RoboDK station: Coursework_2.rdk

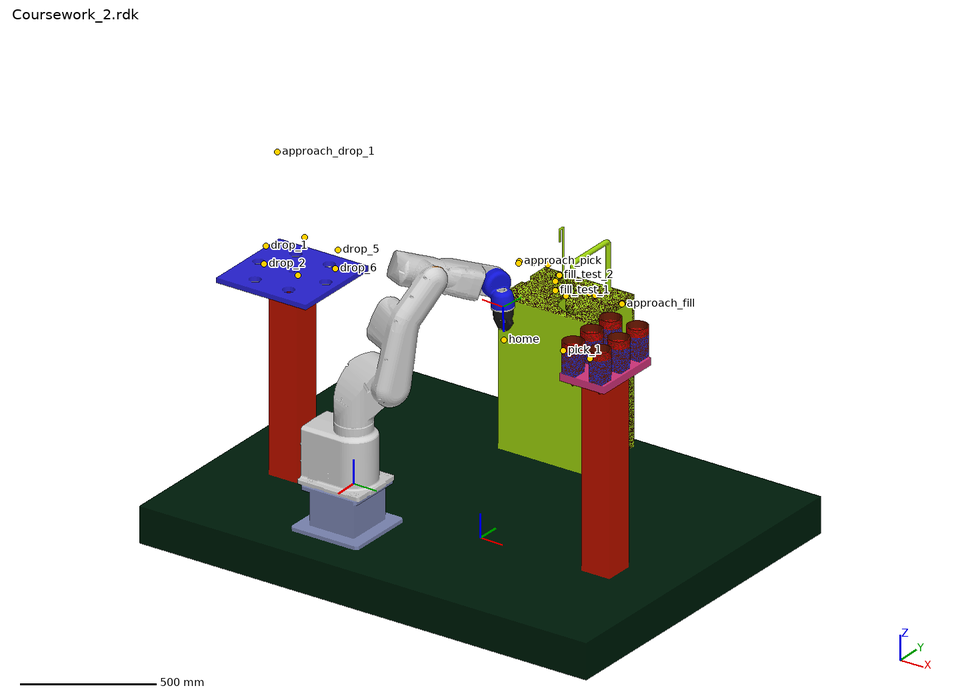
[picture v0: the station drawn from its stored meshes, robots at their saved joint values, targets as dots, program paths as lines]
Station Coursework_2 (saved by RoboDK 5.8.0). Poses are relative to the parent item; angles as X-Y-Z fixed-axis rotations.
Station parameters (name, value as stored): 153.91
  - frame Base_cell_frame at (0, 0, 0) mm
    - object PDE4431_CW2_2024 at (0, 0, 0) mm, rotated rx 90 ry 0 rz 0 deg, size 2000 x 980 x 1500 mm, geometry from PDE4431_CW2_2024.STEP
    - frame Epson VT6 Base at (-250, -450, 330) mm, rotated rx 0 ry 0 rz -90 deg
      - robot Epson VT6: 6 axes, payload 6 kg, reach 920 mm, repeatability 0.1 mm, weight 40 kg
          modified DH rows (alpha deg, a mm, theta deg, d mm): 0, 0, 0, 412; -90, 100, -90, 0; 0, 420, 0, 0; -90, 0, 0, 400; 90, 0, 0, 0; -90, 0, 0, 80
          base shift (0, 0, 0) mm, rotated rx 0 ry 0 rz 90 deg
          joint limits [-170, -160, -51, -200, -125, -360] to [170, 65, 190, 200, 125, 360]; home [0, 0, 0, 0, 0, 0]; saved at [66.458, -23.674, 0.501, 181.108, 64.729, -73.3]
        - frame RobotiQ 2F-140 Gripper (Mechanism) Base at (0, 0, 0) mm
          - robot RobotiQ 2F-140 Gripper (Mechanism) (model RobotiQ 2F140): 1 axes, payload 5 kg
              joint limits [0] to [140]; home [140]; saved at [99.47]
          - target open_gripper (Cartesian target) at (0, 0, 135) mm, rotated rx -90 ry 0 rz 90 deg; joints [99.47, 14.65, 163.72, -0.95, 89.45, -5.12] of RobotiQ 2F-140 Gripper (Mechanism)
          - target close_gripper (Cartesian target) at (0, 0, 135) mm, rotated rx -90 ry 0 rz 90 deg; joints [60, 27.47, -32.86, -122.29, -24.8, -148.93] of RobotiQ 2F-140 Gripper (Mechanism)
        - tool Tool 1, TCP at (0, 0, 135) mm, rotated rx -90 ry 0 rz 90 deg
      - object Pedestal_1 at (0, -30, -180) mm, rotated rx 90 ry 0 rz 0 deg, size 300 x 180 x 300 mm, geometry from Pedestal_1.STEP
    - frame input_table_frame at (0, 0, 0) mm
      - target home (Cartesian target) at (10.77, 139.13, 754.42) mm, rotated rx 88.42 ry -1.71 rz 83.64 deg; joints [-2.51, 19.29, -44.31, 1.89, -63.39, 85.3] of Epson VT6
      - target approach_pick (Cartesian target) at (397.26, -315.09, 1365.72) mm, rotated rx -100.11 ry -87.63 rz -171.58 deg; joints [18.089, -0.789, 29.967, 38.658, -32.785, 56.501] of Epson VT6
      - target pick_1 (Cartesian target) at (594.91, -318.66, 1058.51) mm, rotated rx -100.11 ry -87.63 rz -171.58 deg; joints [7.923, -20.29, 7.849, 146.461, -17.595, -57.734] of Epson VT6
      - target pick_2 (Cartesian target) at (715.78, -319.07, 1058.49) mm, rotated rx -126.16 ry -87.1 rz -145.13 deg; joints [6.525, -37.672, 34.127, 126.782, -9.811, -38.578] of Epson VT6
      - target approach_fill (Cartesian target) at (301.22, 477.28, 847.78) mm, rotated rx -50.46 ry -87.49 rz -131.29 deg; joints [-33.96, -23.408, -22.424, 40.243, 55.613, 64.831] of Epson VT6
      - target enter_fill (Cartesian target) at (181.46, 475.85, 849.63) mm, rotated rx -100.83 ry -88.03 rz -80.88 deg; joints [59.132, -56.563, 37.437, 56.856, 35.551, 37.301] of Epson VT6
      - target fill_1_go_down (Cartesian target) at (99.43, 408.13, 852.78) mm, rotated rx -100.83 ry -88.03 rz -80.88 deg; joints [61.936, -42.802, 12.032, 42.314, 41.214, 54.267] of Epson VT6
      - target fill_test_1 (Cartesian target) at (39.88, 425.07, 848.67) mm, rotated rx -100.83 ry -88.03 rz -80.88 deg; joints [66.768, -41.855, 9.609, 34.939, 39.793, 60.64] of Epson VT6
      - target approach_fill_2 (Cartesian target) at (-3.3, 486.34, 850.99) mm, rotated rx -100.83 ry -88.03 rz -80.88 deg; joints [71.584, -46.813, 19.15, 31.191, 33.677, 62.31] of Epson VT6
      - target fill_2_go_down (Cartesian target) at (-100.56, 579.23, 854.68) mm, rotated rx -100.83 ry -88.03 rz -80.88 deg; joints [79.404, -48.826, 23.503, 18.809, 28.583, 72.676] of Epson VT6
      - target fill_test (Cartesian target) at (-140.12, 595.57, 850.44) mm, rotated rx -100.83 ry -88.03 rz -80.88 deg; joints [82.903, -57.981, 40.297, 15.654, 20.323, 74.725] of Epson VT6
      - target fill_test_3 (Cartesian target) at (-161.01, 566.2, 849.56) mm, rotated rx -100.83 ry -88.03 rz -80.88 deg; joints [84.119, -53.062, 30.713, 10.031, 24.622, 80.354] of Epson VT6
      - target exit_fill (Cartesian target) at (-201.89, 537.42, 848.81) mm, rotated rx -100.83 ry -88.03 rz -80.88 deg; joints [86.913, -48.679, 22.293, 2.884, 28.353, 87.045] of Epson VT6
      - target approach_drop_1 (Cartesian target) at (-801.01, -152.39, 1410.63) mm, rotated rx -121.97 ry -88.27 rz 29.1 deg; joints [139.545, -3.407, 40.97, 127.197, 49.933, -51.748] of Epson VT6
      - target drop_1 (Cartesian target) at (-813.15, -207.69, 1046.6) mm, rotated rx -121.97 ry -88.27 rz 29.1 deg; joints [152.488, 12.57, -28.659, 56.431, 30.004, 35.87] of Epson VT6
      - target drop_2 (Cartesian target) at (-731.62, -336.84, 1047.6) mm, rotated rx -102.73 ry -87.66 rz 14.29 deg; joints [155.972, 28.648, -38.95, 65.094, 28.402, 26.221] of Epson VT6
      - target drop_3 (Cartesian target) at (-739.03, -66.95, 1045.18) mm, rotated rx -102.73 ry -87.66 rz 14.29 deg; joints [125.197, 0.545, -18.808, 75.749, 59.119, 22.393] of Epson VT6
      - target drop_4 (Cartesian target) at (-581.8, -332.78, 1041.64) mm, rotated rx -102.73 ry -87.66 rz 14.29 deg; joints [133.571, 51.579, -47.266, 90.821, 47.936, -4.268] of Epson VT6
      - target drop_5 (Cartesian target) at (-583.93, -72.76, 1039.1) mm, rotated rx -102.73 ry -87.66 rz 14.29 deg; joints [107.283, 10.862, -28.91, 82.785, 75.803, 18.747] of Epson VT6
      - target drop_6 (Cartesian target) at (-505.45, -200.67, 1037.29) mm, rotated rx -102.73 ry -87.66 rz 14.29 deg; joints [99.064, 34.372, -42.989, 86.597, 82.923, 8.461] of Epson VT6
      - target fill_test_2 (Cartesian target) at (-16.95, 531.74, 852.61) mm, rotated rx -100.83 ry -88.03 rz -80.88 deg; joints [73.539, -52.018, 29.199, 32.068, 28.624, 60.312] of Epson VT6
      - target fill_test_4 (Cartesian target) at (166.07, 460.97, 859.21) mm, rotated rx -100.83 ry -88.03 rz -80.88 deg; joints [59.527, -52.804, 31.711, 54.194, 36.359, 40.421] of Epson VT6
      - object Cone_6 at (760, -80, 1030) mm, rotated rx 90 ry 0 rz 0 deg, size 84.9 x 182 x 85 mm, geometry from Cone-Part.STEP
      - object Cone_5 at (640, -80, 1030) mm, rotated rx 90 ry 0 rz 0 deg, size 84.9 x 182 x 85 mm, geometry from Cone-Part.STEP
      - object Cone_4 at (760, -200, 1030) mm, rotated rx 90 ry 0 rz 0 deg, size 84.9 x 182 x 85 mm, geometry from Cone-Part.STEP
      - object Cone_3 at (640, -200, 1030) mm, rotated rx 90 ry 0 rz 0 deg, size 84.9 x 182 x 85 mm, geometry from Cone-Part.STEP
      - object Cone_2 at (760, -320, 1030) mm, rotated rx 90 ry 0 rz 0 deg, size 84.9 x 182 x 85 mm, geometry from Cone-Part.STEP
      - object Cone_1 at (640, -320, 1030) mm, rotated rx 90 ry 0 rz 0 deg, size 84.9 x 182 x 85 mm, geometry from Cone-Part.STEP
  - Python program Main (listed below)
  - program open_gripper (2 instructions, listed below)
  - program close_gripper (2 instructions, listed below)
  - program attach (1 instructions, listed below)
  - program detach (1 instructions, listed below)
  - program replace_1 (1 instructions, listed below)
  - program replace_2 (1 instructions, listed below)
  - program replace_3 (1 instructions, listed below)
  - program replace_4 (1 instructions, listed below)
  - program replace_5 (1 instructions, listed below)
  - program replace_6 (1 instructions, listed below)

--- Python program Main ---
from robodk.robolink import *
from robodk import *
import time
from robodk.robomath import *

RDK = Robolink()  # Establish connection between RoboDK and Python Code
robot = RDK.Item('Epson VT6')
open_gripper_program = RDK.Item('open_gripper', ITEM_TYPE_PROGRAM)  # Opening the gripper
close_gripper_program = RDK.Item('close_gripper', ITEM_TYPE_PROGRAM)  # Closing the gripper
attach = RDK.Item('attach', ITEM_TYPE_PROGRAM)  # Attaching to the gripper
detach = RDK.Item('detach', ITEM_TYPE_PROGRAM)  # Detaching from the gripper
home = RDK.Item('home')

# INPUT STATION - PICKING
pick_1 = RDK.Item('pick_1')
pick_2 = RDK.Item('pick_2')
pick_3 = pick_1.Pose() * transl(0, 0, -120)
pick_4 = pick_2.Pose() * transl(0, 0, -120)
pick_5 = pick_1.Pose() * transl(0, 0, -240)
pick_6 = pick_2.Pose() * transl(0, 0, -240)
approach_pick = RDK.Item('approach_pick')

# FILL STATION (points in order of path)
approach_fill = RDK.Item('approach_fill')
enter_fill = RDK.Item('enter_fill')
fill_test_4 = RDK.Item('fill_test_4')
fill_1_go_down = RDK.Item('fill_1_go_down')
fill_1_go_up = fill_1_go_down.Pose() * transl(15, 0, 0)
fill_test_1 = RDK.Item('fill_test_1')
approach_fill_2 = RDK.Item('approach_fill_2')
fill_test_2 = RDK.Item('fill_test_2')
fill_2_go_down = RDK.Item('fill_2_go_down')
fill_2_go_up = fill_2_go_down.Pose() * transl(15, 0, 0)
exit_fill = RDK.Item('exit_fill')
fill_test = RDK.Item('fill_test')
fill_test_3 = RDK.Item('fill_test_3')

# OUTPUT STATION - DROPPING
approach_drop = RDK.Item('approach_drop')
drop_1 = RDK.Item('drop_1')
drop_2 = RDK.Item('drop_2')
drop_3 = RDK.Item('drop_3')
drop_4 = RDK.Item('drop_4')
drop_5 = RDK.Item('drop_5')
drop_6 = RDK.Item('drop_6')
approach_drop_1 = drop_1.Pose() * transl(100, 0, 0)
approach_drop_2 = drop_2.Pose() * transl(100, 0, 0)
approach_drop_3 = drop_3.Pose() * transl(100, 0, 0)
approach_drop_4 = drop_4.Pose() * transl(100, 0, 0)
approach_drop_5 = drop_5.Pose() * transl(100, 0, 0)
approach_drop_6 = drop_6.Pose() * transl(100, 0, 0)

# Lists for convenience
pick_positions = [pick_1, pick_2, pick_3, pick_4, pick_5, pick_6]
approach_drop_positions = [approach_drop_1, approach_drop_2, approach_drop_3, approach_drop_4, approach_drop_5, approach_drop_6]
drop_positions = [drop_1, drop_2, drop_3, drop_4, drop_5, drop_6]

# Loop through each cone position
for i in range(6):
    # Move to home position and open gripper
    robot.MoveJ(home)
    open_gripper_program.RunProgram()
    time.sleep(1)

    # Move to the approach position and then pick up the cone
    robot.MoveJ(approach_pick)
    robot.MoveL(pick_positions[i])
    time.sleep(1)
    close_gripper_program.RunProgram()
    time.sleep(2)
    attach.RunProgram()
    time.sleep(1)
    robot.MoveL(approach_pick)

    # Move to the filling station
    robot.MoveJ(approach_fill)
    robot.MoveL(enter_fill)

    # Lower speed for filling station
    robot.setSpeed(50)  # Set slower translation speed
    robot.setSpeedJoints(25)  # Set slower joint speed

    # Perform filling operations
    robot.MoveC(fill_test_4, fill_1_go_down)
    robot.MoveL(fill_1_go_up)
    robot.MoveL(fill_1_go_down)
    robot.MoveC(fill_test_1, approach_fill_2)
    robot.MoveC(fill_test_2, fill_2_go_down)
    robot.MoveL(fill_2_go_up)
    robot.MoveL(fill_2_go_down)
    robot.MoveL(fill_test)
    robot.MoveC(fill_test_3, exit_fill)

    # Restore original speed settings
    robot.setSpeed(500)  # Restore translation speed
    robot.setSpeedJoints(150)  # Restore joint speed

    # Move to the dropping station
    robot.MoveL(approach_drop)
    robot.MoveL(approach_drop_positions[i])
    robot.MoveL(drop_positions[i])
    detach.RunProgram()
    time.sleep(1)
    open_gripper_program.RunProgram()  # Open gripper after dropping
    time.sleep(2)
    robot.MoveL(approach_drop_positions[i])  # Go back to approach position

# Finish by moving to home position
time.sleep(1)
robot.MoveJ(home)

--- program open_gripper (robot RobotiQ 2F-140 Gripper (Mechanism)) ---
  Set Ref.: RobotiQ 2F-140 Gripper (Mechanism) Base
  MoveJ (open_gripper)

--- program close_gripper (robot RobotiQ 2F-140 Gripper (Mechanism)) ---
  Set Ref.: RobotiQ 2F-140 Gripper (Mechanism) Base
  MoveJ (close_gripper)

--- program attach (robot Epson VT6) ---
  Attach to Tool 1

--- program detach (robot Epson VT6) ---
  Detach from Tool 1

--- program replace_1 (robot Epson VT6) ---
  Replace objects

--- program replace_2 (robot Epson VT6) ---
  Replace objects

--- program replace_3 (robot Epson VT6) ---
  Replace objects

--- program replace_4 (robot Epson VT6) ---
  Replace objects

--- program replace_5 (robot Epson VT6) ---
  Replace objects

--- program replace_6 (robot Epson VT6) ---
  Replace objects
